// TIA Portal project "BOTTLE" (V18)

(* hardware
DEVICE "S7-300/ET200M station_1"  S7-300 station
   slot 0: "Rail_0"  Rail  6ES7 390-1***0-0AA0
   slot 2: "PLC_1"  CPU 314C-2 DP  6ES7 314-6CG03-0AB0  V2.6
      slot 0: "MPI interface_1"  X1
      slot 1: "DP interface_1"  X2
      slot 2: "DI 24/DO 16_1"  DI24/DO16
      slot 3: "AI 5/AO 2_1"  AI5/AO2
      slot 4: "Count_1"  Counter
      slot 5: "Positioning_1"  Positioning
*)

// ===== PLC "PLC_1"  CPU 314C-2 DP =====

VAR_GLOBAL   // PLC tag table "Tag table_1"
   "step0" AT %M0.0 : Bool;
   "step1" AT %M0.1 : Bool;
   "step2" AT %M0.2 : Bool;
   "step3" AT %M0.3 : Bool;
   "step4" AT %M0.4 : Bool;
   "startbutoon" AT %I125.0 : Bool;
   "cmde_p1" AT %Q124.5 : Bool;
   "cmde_p2" AT %Q124.7 : Bool;
   "cmdr_p1" AT %Q124.6 : Bool;
   "F____S" AT %M0.5 : Bool;
END_VAR

VAR_GLOBAL   // PLC tag table "Default tag table"
   "Tim" AT %M0.6 : Bool;
   "Tim2" AT %M0.7 : Bool;
END_VAR

ORGANIZATION_BLOCK "Main"   // OB1, LAD
TITLE = "Main Program Sweep (Cycle)"
{ S7_Optimized_Access := 'FALSE' }
VERSION : 0.1
   VAR_TEMP
      OB1_EV_CLASS : Byte;   // Bits 0-3 = 1 (Coming event), Bits 4-7 = 1 (Event class 1)
      OB1_SCAN_1 : Byte;   // 1 (Cold restart scan 1 of OB 1), 3 (Scan 2-n of OB 1)
      OB1_PRIORITY : Byte;   // Priority of OB Execution
      OB1_OB_NUMBR : Byte;   // 1 (Organization block 1, OB1)
      OB1_RESERVED_1 : Byte;   // Reserved for system
      OB1_RESERVED_2 : Byte;   // Reserved for system
      OB1_PREV_CYCLE : Int;   // Cycle time of previous OB1 scan (milliseconds)
      OB1_MIN_CYCLE : Int;   // Minimum cycle time of OB1 (milliseconds)
      OB1_MAX_CYCLE : Int;   // Maximum cycle time of OB1 (milliseconds)
      OB1_DATE_TIME : Date_And_Time;   // Date and time OB1 started
   END_VAR
BEGIN

REGION Network 1
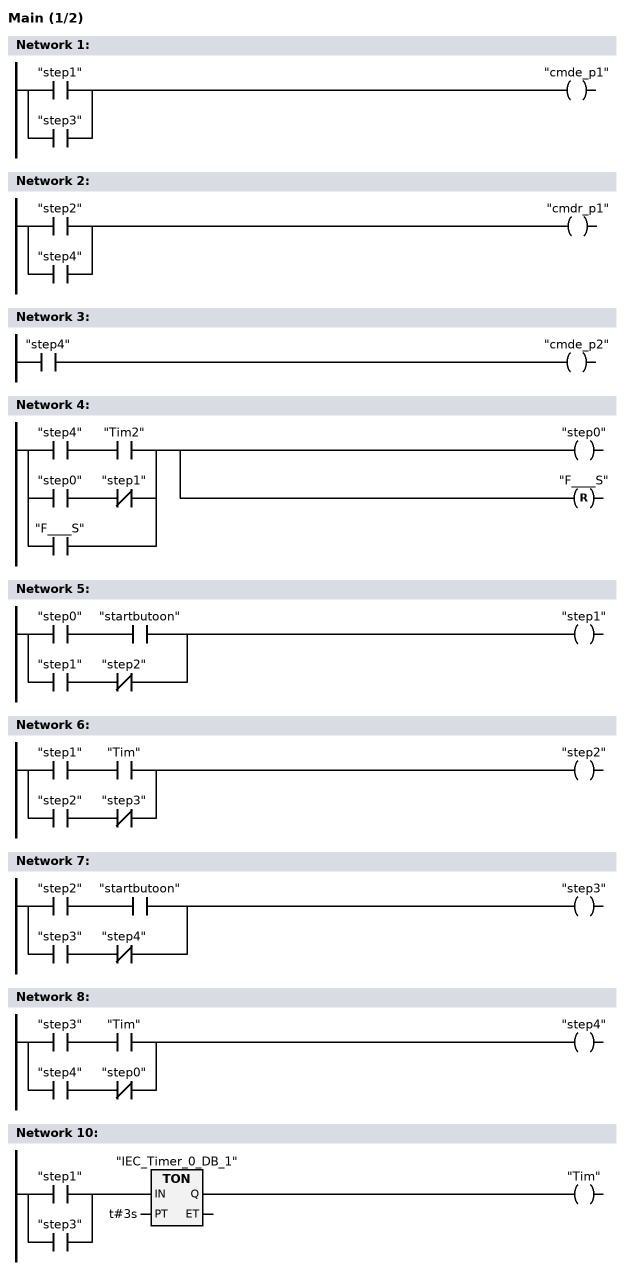
   RUNG wire#powerrail
      Contact( "step1" )
      wire#w1
      Coil( "cmde_p1" )
   END_RUNG
   RUNG wire#powerrail
      Contact( "step3" )
   END_RUNG wire#w1
   // the same network as SCL:
   "cmde_p1" := "step1" OR "step3";
END_REGION

REGION Network 2
   RUNG wire#powerrail
      Contact( "step2" )
      wire#w1
      Coil( "cmdr_p1" )
   END_RUNG
   RUNG wire#powerrail
      Contact( "step4" )
   END_RUNG wire#w1
   // the same network as SCL:
   "cmdr_p1" := "step2" OR "step4";
END_REGION

REGION Network 3
   RUNG wire#powerrail
      Contact( "step4" )
      Coil( "cmde_p2" )
   END_RUNG
   // the same network as SCL:
   "cmde_p2" := "step4";
END_REGION

REGION Network 4
   RUNG wire#powerrail
      Contact( "step4" )
      Contact( "Tim2" )
      wire#w1
      Coil( "step0" )
   END_RUNG
   RUNG wire#powerrail
      Contact( "step0" )
      I_Contact( "step1" )
   END_RUNG wire#w1
   RUNG wire#powerrail
      Contact( "F____S" )
   END_RUNG wire#w1
   RUNG wire#w1
      R_Coil( "F____S" )
   END_RUNG
   // the same network as SCL:
   "step0" := ("step4" AND "Tim2") OR ("step0" AND NOT "step1") OR "F____S";
   IF "step0" THEN "F____S" := FALSE; END_IF;
END_REGION

REGION Network 5
   RUNG wire#powerrail
      Contact( "step0" )
      Contact( "startbutoon" )
      wire#w1
      Coil( "step1" )
   END_RUNG
   RUNG wire#powerrail
      Contact( "step1" )
      I_Contact( "step2" )
   END_RUNG wire#w1
   // the same network as SCL:
   "step1" := ("step0" AND "startbutoon") OR ("step1" AND NOT "step2");
END_REGION

REGION Network 6
   RUNG wire#powerrail
      Contact( "step1" )
      Contact( "Tim" )
      wire#w1
      Coil( "step2" )
   END_RUNG
   RUNG wire#powerrail
      Contact( "step2" )
      I_Contact( "step3" )
   END_RUNG wire#w1
   // the same network as SCL:
   "step2" := ("step1" AND "Tim") OR ("step2" AND NOT "step3");
END_REGION

REGION Network 7
   RUNG wire#powerrail
      Contact( "step2" )
      Contact( "startbutoon" )
      wire#w1
      Coil( "step3" )
   END_RUNG
   RUNG wire#powerrail
      Contact( "step3" )
      I_Contact( "step4" )
   END_RUNG wire#w1
   // the same network as SCL:
   "step3" := ("step2" AND "startbutoon") OR ("step3" AND NOT "step4");
END_REGION

REGION Network 8
   RUNG wire#powerrail
      Contact( "step3" )
      Contact( "Tim" )
      wire#w1
      Coil( "step4" )
   END_RUNG
   RUNG wire#powerrail
      Contact( "step4" )
      I_Contact( "step0" )
   END_RUNG wire#w1
   // the same network as SCL:
   "step4" := ("step3" AND "Tim") OR ("step4" AND NOT "step0");
END_REGION

REGION Network 10
   "IEC_Timer_0_DB_1".TON(IN := "step1" OR "step3", PT := t#3s);
   "Tim" := "IEC_Timer_0_DB_1".Q;
END_REGION

REGION Network 11
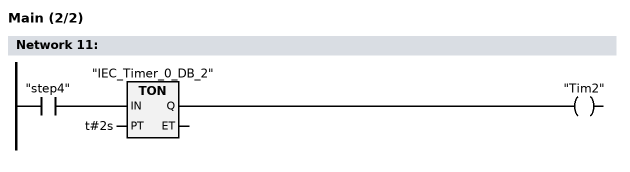
   "IEC_Timer_0_DB_2".TON(IN := "step4", PT := t#2s);
   "Tim2" := "IEC_Timer_0_DB_2".Q;
END_REGION
END_ORGANIZATION_BLOCK

ORGANIZATION_BLOCK "COMPLETE RESTART"   // OB100, LAD
TITLE = "Complete Restart"
{ S7_Optimized_Access := 'FALSE' }
VERSION : 0.1
   VAR_TEMP
      OB100_EV_CLASS : Byte;   // 16#13, Event class 1, Entering event state, Event logged in diagnostic buffer
      OB100_STRTUP : Byte;   // 16#81/82/83/84 Method of startup
      OB100_PRIORITY : Byte;   // Priority of OB Execution
      OB100_OB_NUMBR : Byte;   // 100 (Organization block 100, OB100)
      OB100_RESERVED_1 : Byte;   // Reserved for system
      OB100_RESERVED_2 : Byte;   // Reserved for system
      OB100_STOP : Word;   // Event that caused CPU to stop (16#4xxx)
      OB100_STRT_INFO : DWord;   // Information on how system started
      OB100_DATE_TIME : Date_And_Time;   // Date and time OB100 started
   END_VAR
BEGIN

REGION Network 1
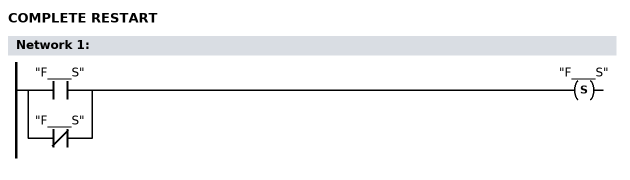
   RUNG wire#powerrail
      Contact( "F____S" )
      wire#w1
      S_Coil( "F____S" )
   END_RUNG
   RUNG wire#powerrail
      I_Contact( "F____S" )
   END_RUNG wire#w1
   // the same network as SCL:
   IF "F____S" OR NOT "F____S" THEN "F____S" := TRUE; END_IF;
END_REGION
END_ORGANIZATION_BLOCK